{attribute 'GeneratedUsingTerminal: EK1122-0000-0018'}
{attribute addProperty BoxType "EK1122-0000-0018"}
{attribute addProperty Id "Beckhoff_EQ3xxxsub_EK1100EK1100_AB5A94672A_0001_EQ3174_0002_0016EQ3174_0E4717A052A_0002_EQ3174_0002_0017EQ3174_0E4717A052A_0003_EQ3174_0002_0021EQ3174_0E4717A052A_0004_EQ3174_0002_0022EQ3174_0E4717A052A_0005_EQ3174_0002_0023EQ3174_0E4717A052A_0006_EQ3204_0002_0016EQ3204_7A00DD1E52A_0007_EQ3204_0002_0017EQ3204_7A00DD1E52A_0008_EQ3204_0002_0020EQ3204_7A00DD1E52A_0009_EQ3204_0002_0021EQ3204_BF0B7ECE48A_0010_EQ3204_0002_0022EQ3204_BF0B7ECE48A_0011_EQ3314_0002_0016EQ3314_CE6B02DE52A_0012_EQ3314_0002_0017EQ3314_CE6B02DE52A_0013_EQ3314_0002_0021EQ3314_CE6B02DE52A_0014_EQ3314_0002_0022EQ3314_6BF23D5548"}
{attribute addProperty CRC "3548460727"}
{attribute addProperty Size "718"}
TYPE Beckhoff_EQ3xxxEK1122_D38136B7 EXTENDS EK1122_AB5A9467 :
STRUCT
	{attribute addProperty Name "Beckhoff_EQ3xxxsub_EK1100"}
	Beckhoff_EQ3xxxsub_EK1100 : EK1100_AB5A9467;
	{attribute addProperty Name "A_0001_EQ3174_0002_0016"}
	A_0001_EQ3174_0002_0016 : EQ3174_0E4717A0;
	{attribute addProperty Name "A_0002_EQ3174_0002_0017"}
	A_0002_EQ3174_0002_0017 : EQ3174_0E4717A0;
	{attribute addProperty Name "A_0003_EQ3174_0002_0021"}
	A_0003_EQ3174_0002_0021 : EQ3174_0E4717A0;
	{attribute addProperty Name "A_0004_EQ3174_0002_0022"}
	A_0004_EQ3174_0002_0022 : EQ3174_0E4717A0;
	{attribute addProperty Name "A_0005_EQ3174_0002_0023"}
	A_0005_EQ3174_0002_0023 : EQ3174_0E4717A0;
	{attribute addProperty Name "A_0006_EQ3204_0002_0016"}
	A_0006_EQ3204_0002_0016 : EQ3204_7A00DD1E;
	{attribute addProperty Name "A_0007_EQ3204_0002_0017"}
	A_0007_EQ3204_0002_0017 : EQ3204_7A00DD1E;
	{attribute addProperty Name "A_0008_EQ3204_0002_0020"}
	A_0008_EQ3204_0002_0020 : EQ3204_7A00DD1E;
	{attribute addProperty Name "A_0009_EQ3204_0002_0021"}
	A_0009_EQ3204_0002_0021 : EQ3204_BF0B7ECE;
	{attribute addProperty Name "A_0010_EQ3204_0002_0022"}
	A_0010_EQ3204_0002_0022 : EQ3204_BF0B7ECE;
	{attribute addProperty Name "A_0011_EQ3314_0002_0016"}
	A_0011_EQ3314_0002_0016 : EQ3314_CE6B02DE;
	{attribute addProperty Name "A_0012_EQ3314_0002_0017"}
	A_0012_EQ3314_0002_0017 : EQ3314_CE6B02DE;
	{attribute addProperty Name "A_0013_EQ3314_0002_0021"}
	A_0013_EQ3314_0002_0021 : EQ3314_CE6B02DE;
	{attribute addProperty Name "A_0014_EQ3314_0002_0022"}
	A_0014_EQ3314_0002_0022 : EQ3314_6BF23D55;
END_STRUCT
END_TYPE

(* stored: Version 1.2.0.0, ProductVersion 3.1.4024.9
   DUT Beckhoff_EQ3xxxEK1122_D38136B7: Id {d2d6307f-4e4e-48ea-9ad4-52764ff07317} *)
